// TIA Portal V20 export
TYPE "UDT_MTP_BinView"
TITLE = MTPDataObjectSUCLibrary/DataAssembly/BinView
   STRUCT
      VState0 { ExternalWritable := 'False'} : String[16] := '';   // Text replacement for false
      VState1 { ExternalWritable := 'False'} : String[16] := '';   // Text replacement for true
      OSLevel : Byte := 16#00;   // OSLevel variable
      WQC { ExternalWritable := 'False'} : Byte := 16#FF;   // Worst Quality code
      V { ExternalWritable := 'False'} : Bool := FALSE;   // Value
   END_STRUCT;
END_TYPE
